// TwinCAT 3 PLC project PLC_Sim
// ProgramVersion: 3.1.4024.0
// libraries:
//   CmpBitmapPool, * (System)
//   Tc2_Standard, * (Beckhoff Automation GmbH)
//   Tc2_System, * (Beckhoff Automation GmbH)
//   Tc3_Module, * (Beckhoff Automation GmbH)
//   VisuSymbols,3.5.10.0,System
// project tree:
//   / GlobalTextList.TcGTLO, PlcTask.TcTTO, Visualization Manager.TcVMO (not stored)
//   GVLs/ GVL.TcGVL
//   POUs/ MAIN.TcPOU, ProcessBlock.TcPOU, Process.TcPOU
//   VISUs/ ImagePool.TcIPO (not stored), Tram.TcVIS (unreadable)

CONFIGURATION PLC_Sim
    RESOURCE PLC ON TwinCAT3
        TASK PlcTask(INTERVAL := T#10ms, PRIORITY := 20);
        PROGRAM MAIN WITH PlcTask : MAIN;
    END_RESOURCE
END_CONFIGURATION

// ---- GVLs/GVL.TcGVL
{attribute 'qualified_only'}
VAR_GLOBAL
	// Input to PLC from process 
	qxSensor1		AT %Q*: BOOL;		(* Sensor at First Station  *)
	qxSensor2		AT %Q*: BOOL;		(* Sensor at Second Station *)
	
	ixButtRight		AT %I*: BOOL;		(* Button for moving the tram Right *)
	ixButtLeft		AT %I*: BOOL;		(* Button for moving the tram Left *)
	
	ixButtManual	AT %I*: BOOL;		(* Button for Manual Mode *)
	ixButtAuto		AT %I*: BOOL;		(* Button for Auto Mode *)
	
	ixButtEmerg     AT %I*: BOOL;		(* Button for Emergency Stop *)
	
	mxSignalRight   AT %I*: BOOL;
	mxSignalLeft    AT %I*: BOOL;
	
	mxAutoRight     AT %I*: BOOL;
	mxAutoLeft      AT %I*: BOOL;
	
	mxEmergRight    AT %I*: BOOL;
	mxEmergLeft     AT %I*: BOOL;
	
	mxEmergManLeft  AT %I*: BOOL;
END_VAR

// ---- POUs/MAIN.TcPOU
PROGRAM MAIN
VAR
END_VAR

Process();

END_PROGRAM

// ---- POUs/Process.TcPOU
PROGRAM Process
VAR
	ProcessBlock_Tram: ProcessBlock;
	ButRight:BOOL;
	ButLeft:BOOL;
END_VAR

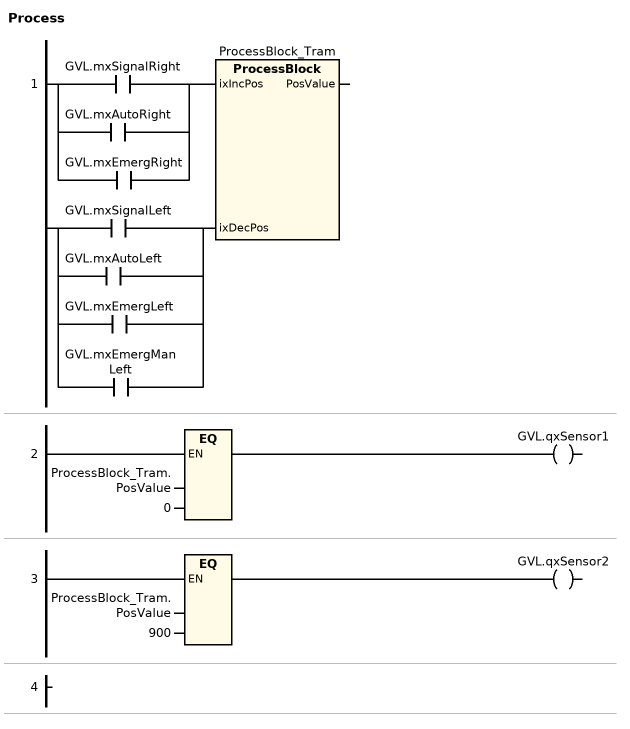
// NETWORK 1
ProcessBlock_Tram(ixIncPos := GVL.mxSignalRight OR GVL.mxAutoRight OR GVL.mxEmergRight, ixDecPos := GVL.mxSignalLeft OR GVL.mxAutoLeft OR GVL.mxEmergLeft OR GVL.mxEmergManLeft); // ProcessBlock

// NETWORK 2
GVL.qxSensor1 := ProcessBlock_Tram.PosValue = 0;

// NETWORK 3
GVL.qxSensor2 := ProcessBlock_Tram.PosValue = 900;

// NETWORK 4

END_PROGRAM

// ---- POUs/ProcessBlock.TcPOU
FUNCTION_BLOCK ProcessBlock
VAR_INPUT
	ixIncPos: BOOL ;
	ixDecPos: BOOL;
END_VAR
VAR_OUTPUT
	PosValue: UINT := 0;
END_VAR
VAR
END_VAR


IF GVL.ixButtManual OR GVL.ixButtAuto THEN
	IF ixIncPos AND PosValue <= 900 AND NOT GVL.qxSensor2 THEN
		IF PosValue > 895 AND PosValue < 900 THEN
			PosValue := 900;
		ELSIF PosValue <= 895 THEN
			PosValue := PosValue + 5;
		END_IF
	END_IF

	IF ixDecPos AND PosValue >= 0 AND NOT GVL.qxSensor1 THEN
		IF PosValue < 5 AND PosValue > 0 THEN
			PosValue := 0;
		ELSIF PosValue >= 5 THEN
			PosValue := PosValue - 5;
		END_IF
	END_IF
END_IF

END_FUNCTION_BLOCK

// ---- GlobalTextList.TcGTLO
TEXTLIST GlobalTextList
  528 = 'Home'
  447 = 'Station 1'
END_TEXTLIST
